// TIA Portal V17 export
// export: Created 2024-08-26T21:07:19.2791777Z, ExportSetting WithDefaults, DisplayName Totally Integrated Automation Portal, DisplayVersion V17 Update 7, DisplayName TIA Portal Openness, DisplayVersion V17 Update 7, DisplayName TIA Portal Version Control Interface, DisplayVersion V17, DisplayName SINAMICS Startdrive Advanced, DisplayVersion V17 SP2, DisplayName SINAMICS Startdrive G110M, G120, G120C, G120D, G120P, G115D, DisplayVersion V17 SP2, DisplayName SINAMICS Startdrive G130, G150, S120, S150, SINAMICS MV, S210, DisplayVersion V17 SP2, DisplayName STEP 7 Professional, DisplayVersion V17 Update 7, DisplayName STEP 7 Safety, DisplayVersion V17 Update 6, DisplayName WinCC Advanced / Unified PC, DisplayVersion V17 Update 7
FUNCTION "DINT TO BOOL" : Void   // FC10, LAD
{ S7_Optimized_Access := 'TRUE' }
VERSION : 0.1
// stored: AutoNumber true, IsIECCheckEnabled false, SetENOAutomatically false, UDAEnableTagReadback false
BEGIN

REGION Network 1: A INPUTS STATUS
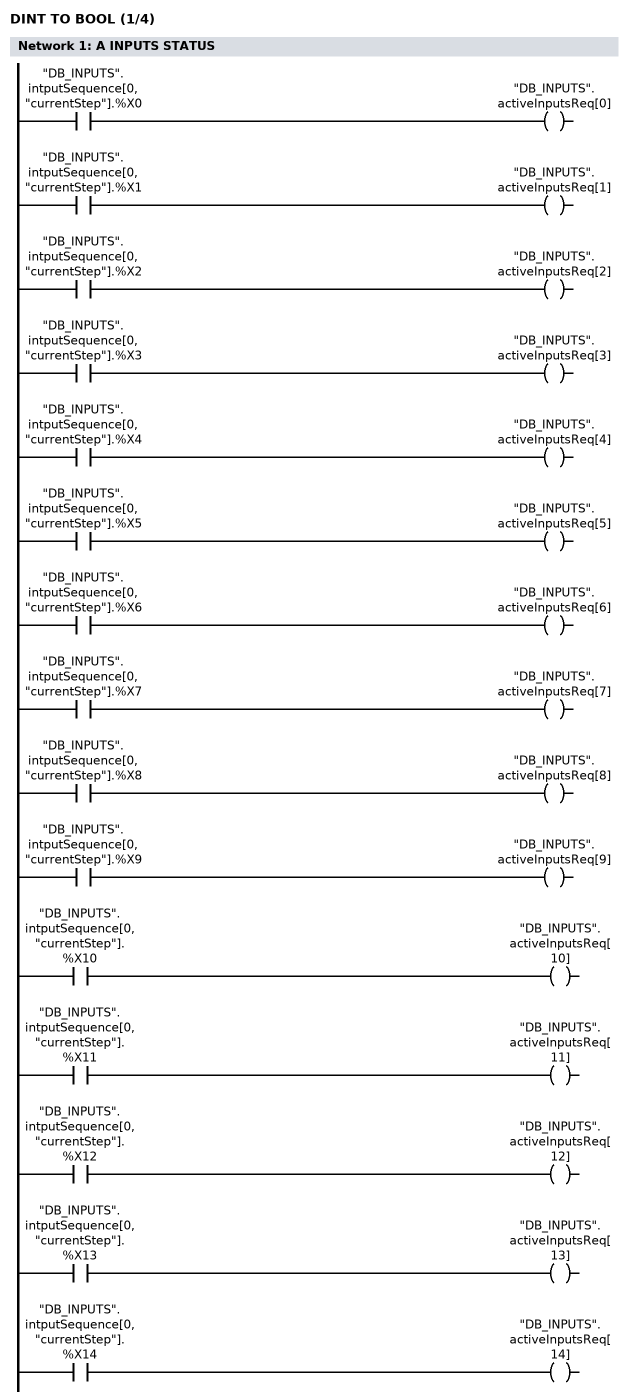
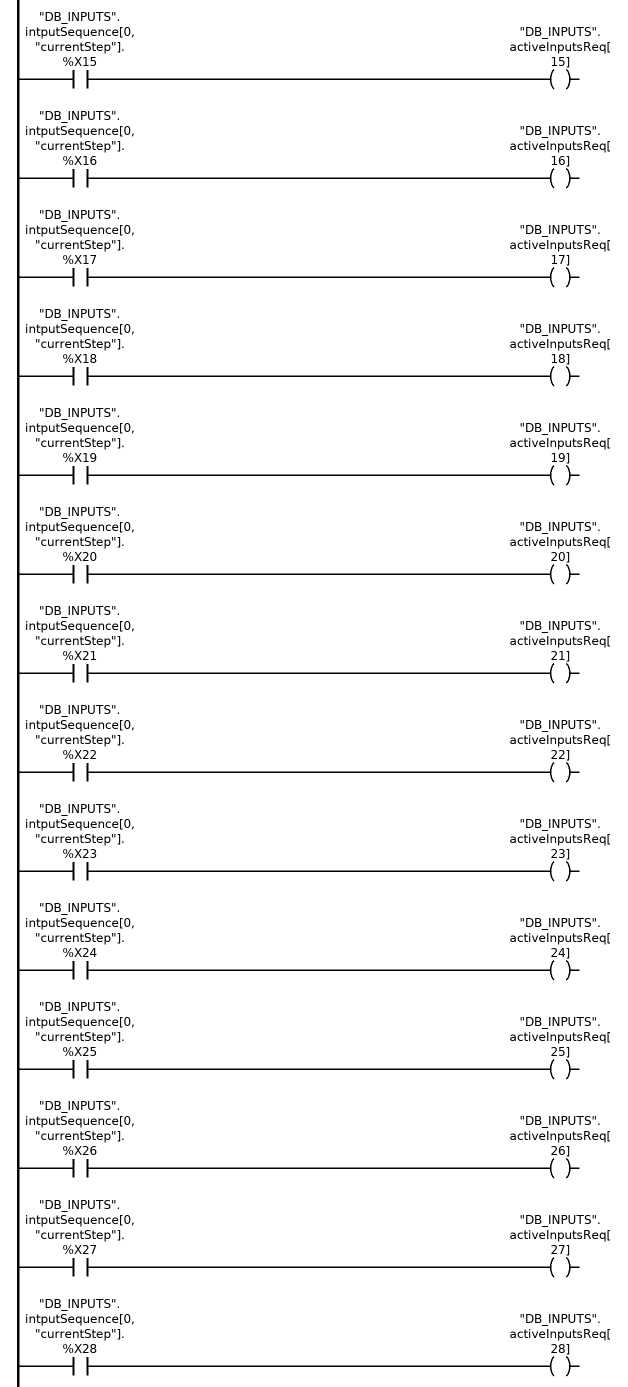
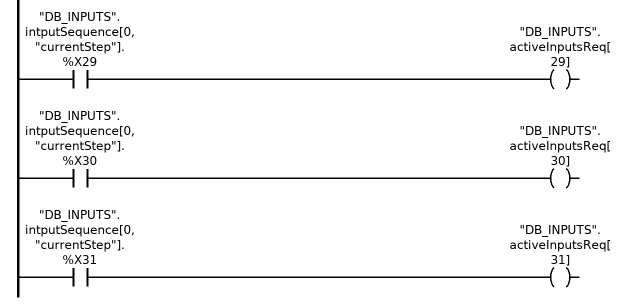
   RUNG wire#powerrail
      Contact( "DB_INPUTS".intputSequence[0, "currentStep"].%X0 )
      Coil( "DB_INPUTS".activeInputsReq[0] )
   END_RUNG
   RUNG wire#powerrail
      Contact( "DB_INPUTS".intputSequence[0, "currentStep"].%X1 )
      Coil( "DB_INPUTS".activeInputsReq[1] )
   END_RUNG
   RUNG wire#powerrail
      Contact( "DB_INPUTS".intputSequence[0, "currentStep"].%X2 )
      Coil( "DB_INPUTS".activeInputsReq[2] )
   END_RUNG
   RUNG wire#powerrail
      Contact( "DB_INPUTS".intputSequence[0, "currentStep"].%X3 )
      Coil( "DB_INPUTS".activeInputsReq[3] )
   END_RUNG
   RUNG wire#powerrail
      Contact( "DB_INPUTS".intputSequence[0, "currentStep"].%X4 )
      Coil( "DB_INPUTS".activeInputsReq[4] )
   END_RUNG
   RUNG wire#powerrail
      Contact( "DB_INPUTS".intputSequence[0, "currentStep"].%X5 )
      Coil( "DB_INPUTS".activeInputsReq[5] )
   END_RUNG
   RUNG wire#powerrail
      Contact( "DB_INPUTS".intputSequence[0, "currentStep"].%X6 )
      Coil( "DB_INPUTS".activeInputsReq[6] )
   END_RUNG
   RUNG wire#powerrail
      Contact( "DB_INPUTS".intputSequence[0, "currentStep"].%X7 )
      Coil( "DB_INPUTS".activeInputsReq[7] )
   END_RUNG
   RUNG wire#powerrail
      Contact( "DB_INPUTS".intputSequence[0, "currentStep"].%X8 )
      Coil( "DB_INPUTS".activeInputsReq[8] )
   END_RUNG
   RUNG wire#powerrail
      Contact( "DB_INPUTS".intputSequence[0, "currentStep"].%X9 )
      Coil( "DB_INPUTS".activeInputsReq[9] )
   END_RUNG
   RUNG wire#powerrail
      Contact( "DB_INPUTS".intputSequence[0, "currentStep"].%X10 )
      Coil( "DB_INPUTS".activeInputsReq[10] )
   END_RUNG
   RUNG wire#powerrail
      Contact( "DB_INPUTS".intputSequence[0, "currentStep"].%X11 )
      Coil( "DB_INPUTS".activeInputsReq[11] )
   END_RUNG
   RUNG wire#powerrail
      Contact( "DB_INPUTS".intputSequence[0, "currentStep"].%X12 )
      Coil( "DB_INPUTS".activeInputsReq[12] )
   END_RUNG
   RUNG wire#powerrail
      Contact( "DB_INPUTS".intputSequence[0, "currentStep"].%X13 )
      Coil( "DB_INPUTS".activeInputsReq[13] )
   END_RUNG
   RUNG wire#powerrail
      Contact( "DB_INPUTS".intputSequence[0, "currentStep"].%X14 )
      Coil( "DB_INPUTS".activeInputsReq[14] )
   END_RUNG
   RUNG wire#powerrail
      Contact( "DB_INPUTS".intputSequence[0, "currentStep"].%X15 )
      Coil( "DB_INPUTS".activeInputsReq[15] )
   END_RUNG
   RUNG wire#powerrail
      Contact( "DB_INPUTS".intputSequence[0, "currentStep"].%X16 )
      Coil( "DB_INPUTS".activeInputsReq[16] )
   END_RUNG
   RUNG wire#powerrail
      Contact( "DB_INPUTS".intputSequence[0, "currentStep"].%X17 )
      Coil( "DB_INPUTS".activeInputsReq[17] )
   END_RUNG
   RUNG wire#powerrail
      Contact( "DB_INPUTS".intputSequence[0, "currentStep"].%X18 )
      Coil( "DB_INPUTS".activeInputsReq[18] )
   END_RUNG
   RUNG wire#powerrail
      Contact( "DB_INPUTS".intputSequence[0, "currentStep"].%X19 )
      Coil( "DB_INPUTS".activeInputsReq[19] )
   END_RUNG
   RUNG wire#powerrail
      Contact( "DB_INPUTS".intputSequence[0, "currentStep"].%X20 )
      Coil( "DB_INPUTS".activeInputsReq[20] )
   END_RUNG
   RUNG wire#powerrail
      Contact( "DB_INPUTS".intputSequence[0, "currentStep"].%X21 )
      Coil( "DB_INPUTS".activeInputsReq[21] )
   END_RUNG
   RUNG wire#powerrail
      Contact( "DB_INPUTS".intputSequence[0, "currentStep"].%X22 )
      Coil( "DB_INPUTS".activeInputsReq[22] )
   END_RUNG
   RUNG wire#powerrail
      Contact( "DB_INPUTS".intputSequence[0, "currentStep"].%X23 )
      Coil( "DB_INPUTS".activeInputsReq[23] )
   END_RUNG
   RUNG wire#powerrail
      Contact( "DB_INPUTS".intputSequence[0, "currentStep"].%X24 )
      Coil( "DB_INPUTS".activeInputsReq[24] )
   END_RUNG
   RUNG wire#powerrail
      Contact( "DB_INPUTS".intputSequence[0, "currentStep"].%X25 )
      Coil( "DB_INPUTS".activeInputsReq[25] )
   END_RUNG
   RUNG wire#powerrail
      Contact( "DB_INPUTS".intputSequence[0, "currentStep"].%X26 )
      Coil( "DB_INPUTS".activeInputsReq[26] )
   END_RUNG
   RUNG wire#powerrail
      Contact( "DB_INPUTS".intputSequence[0, "currentStep"].%X27 )
      Coil( "DB_INPUTS".activeInputsReq[27] )
   END_RUNG
   RUNG wire#powerrail
      Contact( "DB_INPUTS".intputSequence[0, "currentStep"].%X28 )
      Coil( "DB_INPUTS".activeInputsReq[28] )
   END_RUNG
   RUNG wire#powerrail
      Contact( "DB_INPUTS".intputSequence[0, "currentStep"].%X29 )
      Coil( "DB_INPUTS".activeInputsReq[29] )
   END_RUNG
   RUNG wire#powerrail
      Contact( "DB_INPUTS".intputSequence[0, "currentStep"].%X30 )
      Coil( "DB_INPUTS".activeInputsReq[30] )
   END_RUNG
   RUNG wire#powerrail
      Contact( "DB_INPUTS".intputSequence[0, "currentStep"].%X31 )
      Coil( "DB_INPUTS".activeInputsReq[31] )
   END_RUNG
   // the same network as SCL:
   "DB_INPUTS".activeInputsReq[0] := "DB_INPUTS".intputSequence[0, "currentStep"].%X0;
   "DB_INPUTS".activeInputsReq[1] := "DB_INPUTS".intputSequence[0, "currentStep"].%X1;
   "DB_INPUTS".activeInputsReq[2] := "DB_INPUTS".intputSequence[0, "currentStep"].%X2;
   "DB_INPUTS".activeInputsReq[3] := "DB_INPUTS".intputSequence[0, "currentStep"].%X3;
   "DB_INPUTS".activeInputsReq[4] := "DB_INPUTS".intputSequence[0, "currentStep"].%X4;
   "DB_INPUTS".activeInputsReq[5] := "DB_INPUTS".intputSequence[0, "currentStep"].%X5;
   "DB_INPUTS".activeInputsReq[6] := "DB_INPUTS".intputSequence[0, "currentStep"].%X6;
   "DB_INPUTS".activeInputsReq[7] := "DB_INPUTS".intputSequence[0, "currentStep"].%X7;
   "DB_INPUTS".activeInputsReq[8] := "DB_INPUTS".intputSequence[0, "currentStep"].%X8;
   "DB_INPUTS".activeInputsReq[9] := "DB_INPUTS".intputSequence[0, "currentStep"].%X9;
   "DB_INPUTS".activeInputsReq[10] := "DB_INPUTS".intputSequence[0, "currentStep"].%X10;
   "DB_INPUTS".activeInputsReq[11] := "DB_INPUTS".intputSequence[0, "currentStep"].%X11;
   "DB_INPUTS".activeInputsReq[12] := "DB_INPUTS".intputSequence[0, "currentStep"].%X12;
   "DB_INPUTS".activeInputsReq[13] := "DB_INPUTS".intputSequence[0, "currentStep"].%X13;
   "DB_INPUTS".activeInputsReq[14] := "DB_INPUTS".intputSequence[0, "currentStep"].%X14;
   "DB_INPUTS".activeInputsReq[15] := "DB_INPUTS".intputSequence[0, "currentStep"].%X15;
   "DB_INPUTS".activeInputsReq[16] := "DB_INPUTS".intputSequence[0, "currentStep"].%X16;
   "DB_INPUTS".activeInputsReq[17] := "DB_INPUTS".intputSequence[0, "currentStep"].%X17;
   "DB_INPUTS".activeInputsReq[18] := "DB_INPUTS".intputSequence[0, "currentStep"].%X18;
   "DB_INPUTS".activeInputsReq[19] := "DB_INPUTS".intputSequence[0, "currentStep"].%X19;
   "DB_INPUTS".activeInputsReq[20] := "DB_INPUTS".intputSequence[0, "currentStep"].%X20;
   "DB_INPUTS".activeInputsReq[21] := "DB_INPUTS".intputSequence[0, "currentStep"].%X21;
   "DB_INPUTS".activeInputsReq[22] := "DB_INPUTS".intputSequence[0, "currentStep"].%X22;
   "DB_INPUTS".activeInputsReq[23] := "DB_INPUTS".intputSequence[0, "currentStep"].%X23;
   "DB_INPUTS".activeInputsReq[24] := "DB_INPUTS".intputSequence[0, "currentStep"].%X24;
   "DB_INPUTS".activeInputsReq[25] := "DB_INPUTS".intputSequence[0, "currentStep"].%X25;
   "DB_INPUTS".activeInputsReq[26] := "DB_INPUTS".intputSequence[0, "currentStep"].%X26;
   "DB_INPUTS".activeInputsReq[27] := "DB_INPUTS".intputSequence[0, "currentStep"].%X27;
   "DB_INPUTS".activeInputsReq[28] := "DB_INPUTS".intputSequence[0, "currentStep"].%X28;
   "DB_INPUTS".activeInputsReq[29] := "DB_INPUTS".intputSequence[0, "currentStep"].%X29;
   "DB_INPUTS".activeInputsReq[30] := "DB_INPUTS".intputSequence[0, "currentStep"].%X30;
   "DB_INPUTS".activeInputsReq[31] := "DB_INPUTS".intputSequence[0, "currentStep"].%X31;
END_REGION

REGION Network 2: MASK INPUTS STATUS
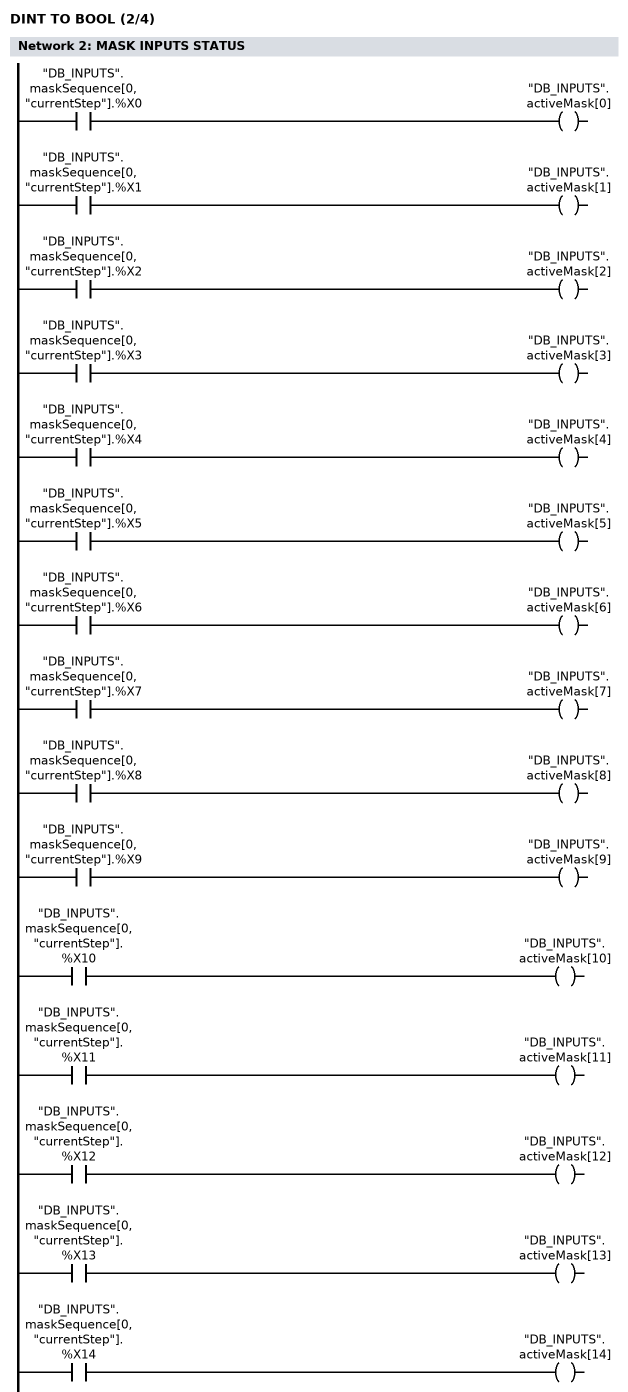
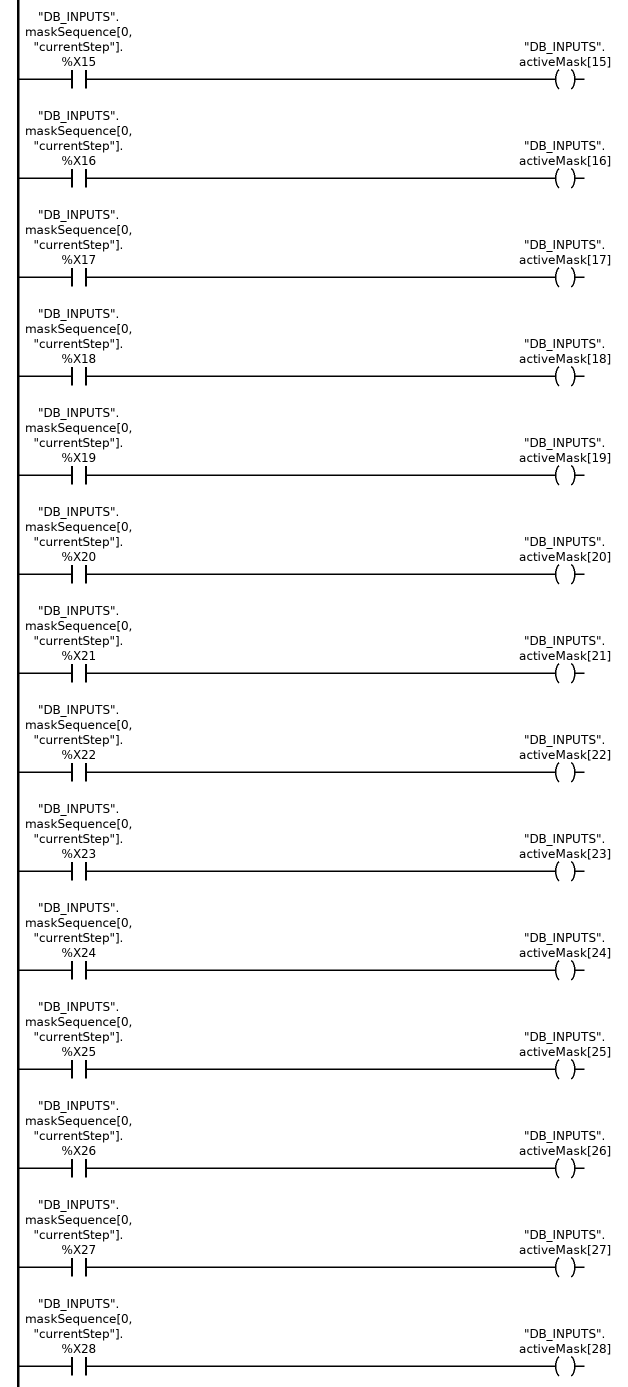
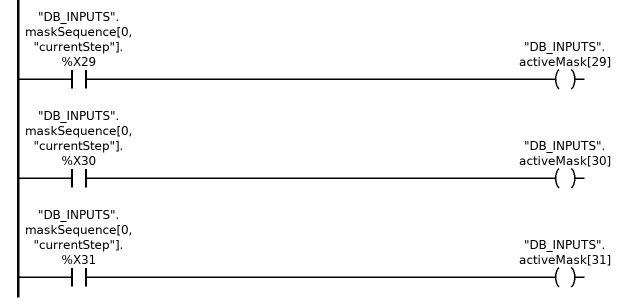
   RUNG wire#powerrail
      Contact( "DB_INPUTS".maskSequence[0, "currentStep"].%X0 )
      Coil( "DB_INPUTS".activeMask[0] )
   END_RUNG
   RUNG wire#powerrail
      Contact( "DB_INPUTS".maskSequence[0, "currentStep"].%X1 )
      Coil( "DB_INPUTS".activeMask[1] )
   END_RUNG
   RUNG wire#powerrail
      Contact( "DB_INPUTS".maskSequence[0, "currentStep"].%X2 )
      Coil( "DB_INPUTS".activeMask[2] )
   END_RUNG
   RUNG wire#powerrail
      Contact( "DB_INPUTS".maskSequence[0, "currentStep"].%X3 )
      Coil( "DB_INPUTS".activeMask[3] )
   END_RUNG
   RUNG wire#powerrail
      Contact( "DB_INPUTS".maskSequence[0, "currentStep"].%X4 )
      Coil( "DB_INPUTS".activeMask[4] )
   END_RUNG
   RUNG wire#powerrail
      Contact( "DB_INPUTS".maskSequence[0, "currentStep"].%X5 )
      Coil( "DB_INPUTS".activeMask[5] )
   END_RUNG
   RUNG wire#powerrail
      Contact( "DB_INPUTS".maskSequence[0, "currentStep"].%X6 )
      Coil( "DB_INPUTS".activeMask[6] )
   END_RUNG
   RUNG wire#powerrail
      Contact( "DB_INPUTS".maskSequence[0, "currentStep"].%X7 )
      Coil( "DB_INPUTS".activeMask[7] )
   END_RUNG
   RUNG wire#powerrail
      Contact( "DB_INPUTS".maskSequence[0, "currentStep"].%X8 )
      Coil( "DB_INPUTS".activeMask[8] )
   END_RUNG
   RUNG wire#powerrail
      Contact( "DB_INPUTS".maskSequence[0, "currentStep"].%X9 )
      Coil( "DB_INPUTS".activeMask[9] )
   END_RUNG
   RUNG wire#powerrail
      Contact( "DB_INPUTS".maskSequence[0, "currentStep"].%X10 )
      Coil( "DB_INPUTS".activeMask[10] )
   END_RUNG
   RUNG wire#powerrail
      Contact( "DB_INPUTS".maskSequence[0, "currentStep"].%X11 )
      Coil( "DB_INPUTS".activeMask[11] )
   END_RUNG
   RUNG wire#powerrail
      Contact( "DB_INPUTS".maskSequence[0, "currentStep"].%X12 )
      Coil( "DB_INPUTS".activeMask[12] )
   END_RUNG
   RUNG wire#powerrail
      Contact( "DB_INPUTS".maskSequence[0, "currentStep"].%X13 )
      Coil( "DB_INPUTS".activeMask[13] )
   END_RUNG
   RUNG wire#powerrail
      Contact( "DB_INPUTS".maskSequence[0, "currentStep"].%X14 )
      Coil( "DB_INPUTS".activeMask[14] )
   END_RUNG
   RUNG wire#powerrail
      Contact( "DB_INPUTS".maskSequence[0, "currentStep"].%X15 )
      Coil( "DB_INPUTS".activeMask[15] )
   END_RUNG
   RUNG wire#powerrail
      Contact( "DB_INPUTS".maskSequence[0, "currentStep"].%X16 )
      Coil( "DB_INPUTS".activeMask[16] )
   END_RUNG
   RUNG wire#powerrail
      Contact( "DB_INPUTS".maskSequence[0, "currentStep"].%X17 )
      Coil( "DB_INPUTS".activeMask[17] )
   END_RUNG
   RUNG wire#powerrail
      Contact( "DB_INPUTS".maskSequence[0, "currentStep"].%X18 )
      Coil( "DB_INPUTS".activeMask[18] )
   END_RUNG
   RUNG wire#powerrail
      Contact( "DB_INPUTS".maskSequence[0, "currentStep"].%X19 )
      Coil( "DB_INPUTS".activeMask[19] )
   END_RUNG
   RUNG wire#powerrail
      Contact( "DB_INPUTS".maskSequence[0, "currentStep"].%X20 )
      Coil( "DB_INPUTS".activeMask[20] )
   END_RUNG
   RUNG wire#powerrail
      Contact( "DB_INPUTS".maskSequence[0, "currentStep"].%X21 )
      Coil( "DB_INPUTS".activeMask[21] )
   END_RUNG
   RUNG wire#powerrail
      Contact( "DB_INPUTS".maskSequence[0, "currentStep"].%X22 )
      Coil( "DB_INPUTS".activeMask[22] )
   END_RUNG
   RUNG wire#powerrail
      Contact( "DB_INPUTS".maskSequence[0, "currentStep"].%X23 )
      Coil( "DB_INPUTS".activeMask[23] )
   END_RUNG
   RUNG wire#powerrail
      Contact( "DB_INPUTS".maskSequence[0, "currentStep"].%X24 )
      Coil( "DB_INPUTS".activeMask[24] )
   END_RUNG
   RUNG wire#powerrail
      Contact( "DB_INPUTS".maskSequence[0, "currentStep"].%X25 )
      Coil( "DB_INPUTS".activeMask[25] )
   END_RUNG
   RUNG wire#powerrail
      Contact( "DB_INPUTS".maskSequence[0, "currentStep"].%X26 )
      Coil( "DB_INPUTS".activeMask[26] )
   END_RUNG
   RUNG wire#powerrail
      Contact( "DB_INPUTS".maskSequence[0, "currentStep"].%X27 )
      Coil( "DB_INPUTS".activeMask[27] )
   END_RUNG
   RUNG wire#powerrail
      Contact( "DB_INPUTS".maskSequence[0, "currentStep"].%X28 )
      Coil( "DB_INPUTS".activeMask[28] )
   END_RUNG
   RUNG wire#powerrail
      Contact( "DB_INPUTS".maskSequence[0, "currentStep"].%X29 )
      Coil( "DB_INPUTS".activeMask[29] )
   END_RUNG
   RUNG wire#powerrail
      Contact( "DB_INPUTS".maskSequence[0, "currentStep"].%X30 )
      Coil( "DB_INPUTS".activeMask[30] )
   END_RUNG
   RUNG wire#powerrail
      Contact( "DB_INPUTS".maskSequence[0, "currentStep"].%X31 )
      Coil( "DB_INPUTS".activeMask[31] )
   END_RUNG
   // the same network as SCL:
   "DB_INPUTS".activeMask[0] := "DB_INPUTS".maskSequence[0, "currentStep"].%X0;
   "DB_INPUTS".activeMask[1] := "DB_INPUTS".maskSequence[0, "currentStep"].%X1;
   "DB_INPUTS".activeMask[2] := "DB_INPUTS".maskSequence[0, "currentStep"].%X2;
   "DB_INPUTS".activeMask[3] := "DB_INPUTS".maskSequence[0, "currentStep"].%X3;
   "DB_INPUTS".activeMask[4] := "DB_INPUTS".maskSequence[0, "currentStep"].%X4;
   "DB_INPUTS".activeMask[5] := "DB_INPUTS".maskSequence[0, "currentStep"].%X5;
   "DB_INPUTS".activeMask[6] := "DB_INPUTS".maskSequence[0, "currentStep"].%X6;
   "DB_INPUTS".activeMask[7] := "DB_INPUTS".maskSequence[0, "currentStep"].%X7;
   "DB_INPUTS".activeMask[8] := "DB_INPUTS".maskSequence[0, "currentStep"].%X8;
   "DB_INPUTS".activeMask[9] := "DB_INPUTS".maskSequence[0, "currentStep"].%X9;
   "DB_INPUTS".activeMask[10] := "DB_INPUTS".maskSequence[0, "currentStep"].%X10;
   "DB_INPUTS".activeMask[11] := "DB_INPUTS".maskSequence[0, "currentStep"].%X11;
   "DB_INPUTS".activeMask[12] := "DB_INPUTS".maskSequence[0, "currentStep"].%X12;
   "DB_INPUTS".activeMask[13] := "DB_INPUTS".maskSequence[0, "currentStep"].%X13;
   "DB_INPUTS".activeMask[14] := "DB_INPUTS".maskSequence[0, "currentStep"].%X14;
   "DB_INPUTS".activeMask[15] := "DB_INPUTS".maskSequence[0, "currentStep"].%X15;
   "DB_INPUTS".activeMask[16] := "DB_INPUTS".maskSequence[0, "currentStep"].%X16;
   "DB_INPUTS".activeMask[17] := "DB_INPUTS".maskSequence[0, "currentStep"].%X17;
   "DB_INPUTS".activeMask[18] := "DB_INPUTS".maskSequence[0, "currentStep"].%X18;
   "DB_INPUTS".activeMask[19] := "DB_INPUTS".maskSequence[0, "currentStep"].%X19;
   "DB_INPUTS".activeMask[20] := "DB_INPUTS".maskSequence[0, "currentStep"].%X20;
   "DB_INPUTS".activeMask[21] := "DB_INPUTS".maskSequence[0, "currentStep"].%X21;
   "DB_INPUTS".activeMask[22] := "DB_INPUTS".maskSequence[0, "currentStep"].%X22;
   "DB_INPUTS".activeMask[23] := "DB_INPUTS".maskSequence[0, "currentStep"].%X23;
   "DB_INPUTS".activeMask[24] := "DB_INPUTS".maskSequence[0, "currentStep"].%X24;
   "DB_INPUTS".activeMask[25] := "DB_INPUTS".maskSequence[0, "currentStep"].%X25;
   "DB_INPUTS".activeMask[26] := "DB_INPUTS".maskSequence[0, "currentStep"].%X26;
   "DB_INPUTS".activeMask[27] := "DB_INPUTS".maskSequence[0, "currentStep"].%X27;
   "DB_INPUTS".activeMask[28] := "DB_INPUTS".maskSequence[0, "currentStep"].%X28;
   "DB_INPUTS".activeMask[29] := "DB_INPUTS".maskSequence[0, "currentStep"].%X29;
   "DB_INPUTS".activeMask[30] := "DB_INPUTS".maskSequence[0, "currentStep"].%X30;
   "DB_INPUTS".activeMask[31] := "DB_INPUTS".maskSequence[0, "currentStep"].%X31;
END_REGION

REGION Network 3: B OUTPUTS STATUS
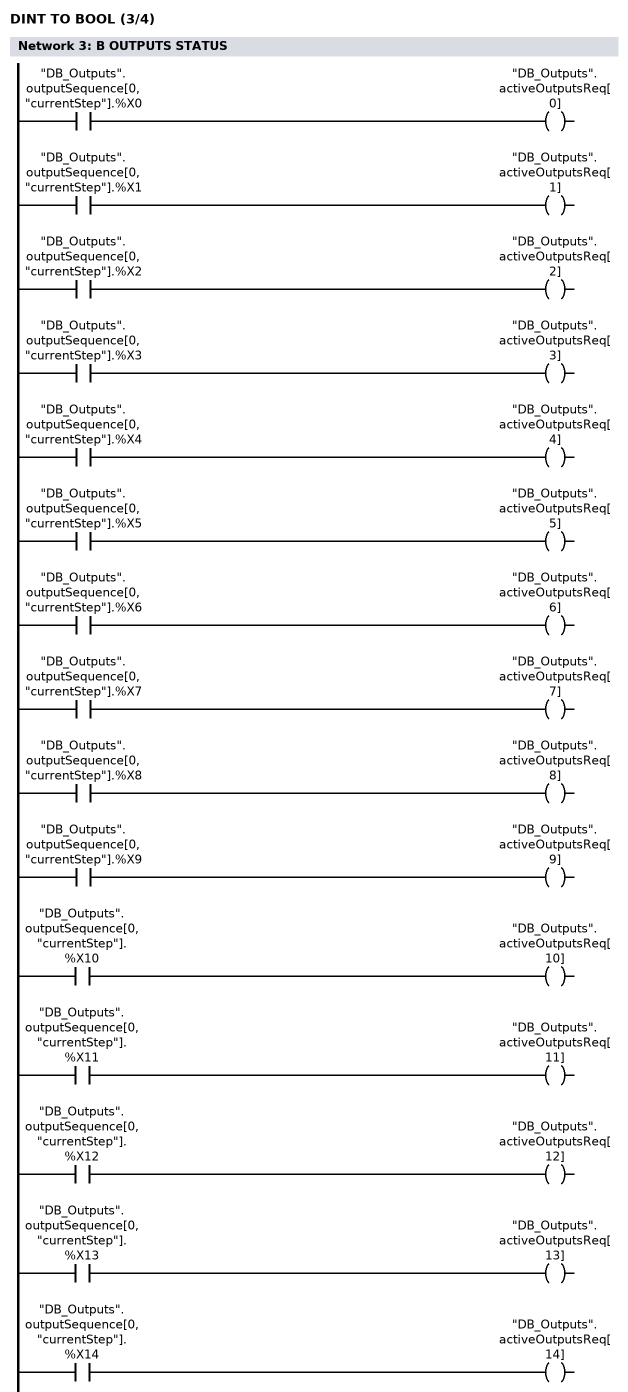
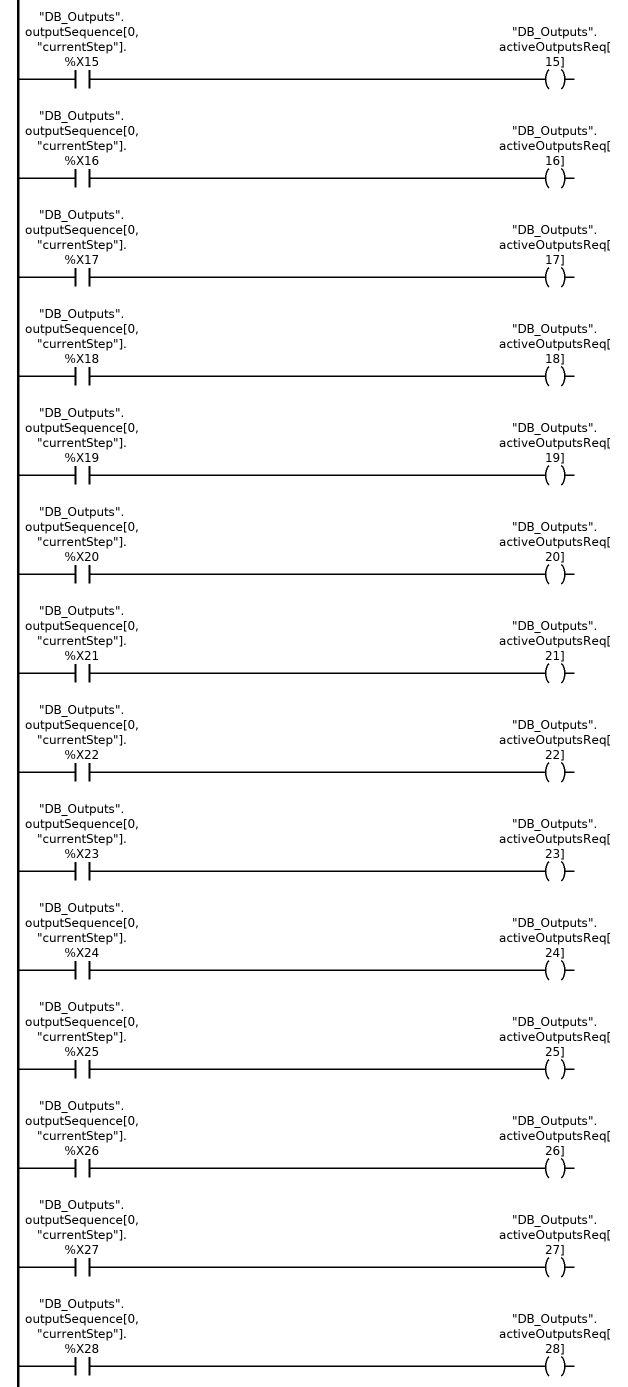
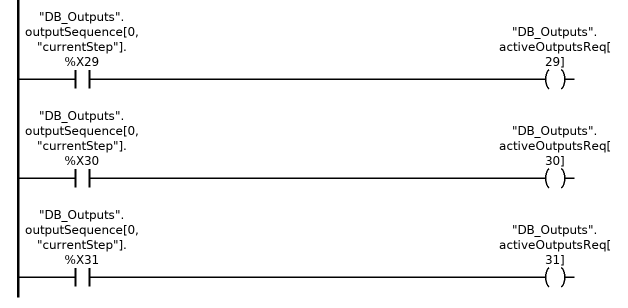
   RUNG wire#powerrail
      Contact( "DB_Outputs".outputSequence[0, "currentStep"].%X0 )
      Coil( "DB_Outputs".activeOutputsReq[0] )
   END_RUNG
   RUNG wire#powerrail
      Contact( "DB_Outputs".outputSequence[0, "currentStep"].%X1 )
      Coil( "DB_Outputs".activeOutputsReq[1] )
   END_RUNG
   RUNG wire#powerrail
      Contact( "DB_Outputs".outputSequence[0, "currentStep"].%X2 )
      Coil( "DB_Outputs".activeOutputsReq[2] )
   END_RUNG
   RUNG wire#powerrail
      Contact( "DB_Outputs".outputSequence[0, "currentStep"].%X3 )
      Coil( "DB_Outputs".activeOutputsReq[3] )
   END_RUNG
   RUNG wire#powerrail
      Contact( "DB_Outputs".outputSequence[0, "currentStep"].%X4 )
      Coil( "DB_Outputs".activeOutputsReq[4] )
   END_RUNG
   RUNG wire#powerrail
      Contact( "DB_Outputs".outputSequence[0, "currentStep"].%X5 )
      Coil( "DB_Outputs".activeOutputsReq[5] )
   END_RUNG
   RUNG wire#powerrail
      Contact( "DB_Outputs".outputSequence[0, "currentStep"].%X6 )
      Coil( "DB_Outputs".activeOutputsReq[6] )
   END_RUNG
   RUNG wire#powerrail
      Contact( "DB_Outputs".outputSequence[0, "currentStep"].%X7 )
      Coil( "DB_Outputs".activeOutputsReq[7] )
   END_RUNG
   RUNG wire#powerrail
      Contact( "DB_Outputs".outputSequence[0, "currentStep"].%X8 )
      Coil( "DB_Outputs".activeOutputsReq[8] )
   END_RUNG
   RUNG wire#powerrail
      Contact( "DB_Outputs".outputSequence[0, "currentStep"].%X9 )
      Coil( "DB_Outputs".activeOutputsReq[9] )
   END_RUNG
   RUNG wire#powerrail
      Contact( "DB_Outputs".outputSequence[0, "currentStep"].%X10 )
      Coil( "DB_Outputs".activeOutputsReq[10] )
   END_RUNG
   RUNG wire#powerrail
      Contact( "DB_Outputs".outputSequence[0, "currentStep"].%X11 )
      Coil( "DB_Outputs".activeOutputsReq[11] )
   END_RUNG
   RUNG wire#powerrail
      Contact( "DB_Outputs".outputSequence[0, "currentStep"].%X12 )
      Coil( "DB_Outputs".activeOutputsReq[12] )
   END_RUNG
   RUNG wire#powerrail
      Contact( "DB_Outputs".outputSequence[0, "currentStep"].%X13 )
      Coil( "DB_Outputs".activeOutputsReq[13] )
   END_RUNG
   RUNG wire#powerrail
      Contact( "DB_Outputs".outputSequence[0, "currentStep"].%X14 )
      Coil( "DB_Outputs".activeOutputsReq[14] )
   END_RUNG
   RUNG wire#powerrail
      Contact( "DB_Outputs".outputSequence[0, "currentStep"].%X15 )
      Coil( "DB_Outputs".activeOutputsReq[15] )
   END_RUNG
   RUNG wire#powerrail
      Contact( "DB_Outputs".outputSequence[0, "currentStep"].%X16 )
      Coil( "DB_Outputs".activeOutputsReq[16] )
   END_RUNG
   RUNG wire#powerrail
      Contact( "DB_Outputs".outputSequence[0, "currentStep"].%X17 )
      Coil( "DB_Outputs".activeOutputsReq[17] )
   END_RUNG
   RUNG wire#powerrail
      Contact( "DB_Outputs".outputSequence[0, "currentStep"].%X18 )
      Coil( "DB_Outputs".activeOutputsReq[18] )
   END_RUNG
   RUNG wire#powerrail
      Contact( "DB_Outputs".outputSequence[0, "currentStep"].%X19 )
      Coil( "DB_Outputs".activeOutputsReq[19] )
   END_RUNG
   RUNG wire#powerrail
      Contact( "DB_Outputs".outputSequence[0, "currentStep"].%X20 )
      Coil( "DB_Outputs".activeOutputsReq[20] )
   END_RUNG
   RUNG wire#powerrail
      Contact( "DB_Outputs".outputSequence[0, "currentStep"].%X21 )
      Coil( "DB_Outputs".activeOutputsReq[21] )
   END_RUNG
   RUNG wire#powerrail
      Contact( "DB_Outputs".outputSequence[0, "currentStep"].%X22 )
      Coil( "DB_Outputs".activeOutputsReq[22] )
   END_RUNG
   RUNG wire#powerrail
      Contact( "DB_Outputs".outputSequence[0, "currentStep"].%X23 )
      Coil( "DB_Outputs".activeOutputsReq[23] )
   END_RUNG
   RUNG wire#powerrail
      Contact( "DB_Outputs".outputSequence[0, "currentStep"].%X24 )
      Coil( "DB_Outputs".activeOutputsReq[24] )
   END_RUNG
   RUNG wire#powerrail
      Contact( "DB_Outputs".outputSequence[0, "currentStep"].%X25 )
      Coil( "DB_Outputs".activeOutputsReq[25] )
   END_RUNG
   RUNG wire#powerrail
      Contact( "DB_Outputs".outputSequence[0, "currentStep"].%X26 )
      Coil( "DB_Outputs".activeOutputsReq[26] )
   END_RUNG
   RUNG wire#powerrail
      Contact( "DB_Outputs".outputSequence[0, "currentStep"].%X27 )
      Coil( "DB_Outputs".activeOutputsReq[27] )
   END_RUNG
   RUNG wire#powerrail
      Contact( "DB_Outputs".outputSequence[0, "currentStep"].%X28 )
      Coil( "DB_Outputs".activeOutputsReq[28] )
   END_RUNG
   RUNG wire#powerrail
      Contact( "DB_Outputs".outputSequence[0, "currentStep"].%X29 )
      Coil( "DB_Outputs".activeOutputsReq[29] )
   END_RUNG
   RUNG wire#powerrail
      Contact( "DB_Outputs".outputSequence[0, "currentStep"].%X30 )
      Coil( "DB_Outputs".activeOutputsReq[30] )
   END_RUNG
   RUNG wire#powerrail
      Contact( "DB_Outputs".outputSequence[0, "currentStep"].%X31 )
      Coil( "DB_Outputs".activeOutputsReq[31] )
   END_RUNG
   // the same network as SCL:
   "DB_Outputs".activeOutputsReq[0] := "DB_Outputs".outputSequence[0, "currentStep"].%X0;
   "DB_Outputs".activeOutputsReq[1] := "DB_Outputs".outputSequence[0, "currentStep"].%X1;
   "DB_Outputs".activeOutputsReq[2] := "DB_Outputs".outputSequence[0, "currentStep"].%X2;
   "DB_Outputs".activeOutputsReq[3] := "DB_Outputs".outputSequence[0, "currentStep"].%X3;
   "DB_Outputs".activeOutputsReq[4] := "DB_Outputs".outputSequence[0, "currentStep"].%X4;
   "DB_Outputs".activeOutputsReq[5] := "DB_Outputs".outputSequence[0, "currentStep"].%X5;
   "DB_Outputs".activeOutputsReq[6] := "DB_Outputs".outputSequence[0, "currentStep"].%X6;
   "DB_Outputs".activeOutputsReq[7] := "DB_Outputs".outputSequence[0, "currentStep"].%X7;
   "DB_Outputs".activeOutputsReq[8] := "DB_Outputs".outputSequence[0, "currentStep"].%X8;
   "DB_Outputs".activeOutputsReq[9] := "DB_Outputs".outputSequence[0, "currentStep"].%X9;
   "DB_Outputs".activeOutputsReq[10] := "DB_Outputs".outputSequence[0, "currentStep"].%X10;
   "DB_Outputs".activeOutputsReq[11] := "DB_Outputs".outputSequence[0, "currentStep"].%X11;
   "DB_Outputs".activeOutputsReq[12] := "DB_Outputs".outputSequence[0, "currentStep"].%X12;
   "DB_Outputs".activeOutputsReq[13] := "DB_Outputs".outputSequence[0, "currentStep"].%X13;
   "DB_Outputs".activeOutputsReq[14] := "DB_Outputs".outputSequence[0, "currentStep"].%X14;
   "DB_Outputs".activeOutputsReq[15] := "DB_Outputs".outputSequence[0, "currentStep"].%X15;
   "DB_Outputs".activeOutputsReq[16] := "DB_Outputs".outputSequence[0, "currentStep"].%X16;
   "DB_Outputs".activeOutputsReq[17] := "DB_Outputs".outputSequence[0, "currentStep"].%X17;
   "DB_Outputs".activeOutputsReq[18] := "DB_Outputs".outputSequence[0, "currentStep"].%X18;
   "DB_Outputs".activeOutputsReq[19] := "DB_Outputs".outputSequence[0, "currentStep"].%X19;
   "DB_Outputs".activeOutputsReq[20] := "DB_Outputs".outputSequence[0, "currentStep"].%X20;
   "DB_Outputs".activeOutputsReq[21] := "DB_Outputs".outputSequence[0, "currentStep"].%X21;
   "DB_Outputs".activeOutputsReq[22] := "DB_Outputs".outputSequence[0, "currentStep"].%X22;
   "DB_Outputs".activeOutputsReq[23] := "DB_Outputs".outputSequence[0, "currentStep"].%X23;
   "DB_Outputs".activeOutputsReq[24] := "DB_Outputs".outputSequence[0, "currentStep"].%X24;
   "DB_Outputs".activeOutputsReq[25] := "DB_Outputs".outputSequence[0, "currentStep"].%X25;
   "DB_Outputs".activeOutputsReq[26] := "DB_Outputs".outputSequence[0, "currentStep"].%X26;
   "DB_Outputs".activeOutputsReq[27] := "DB_Outputs".outputSequence[0, "currentStep"].%X27;
   "DB_Outputs".activeOutputsReq[28] := "DB_Outputs".outputSequence[0, "currentStep"].%X28;
   "DB_Outputs".activeOutputsReq[29] := "DB_Outputs".outputSequence[0, "currentStep"].%X29;
   "DB_Outputs".activeOutputsReq[30] := "DB_Outputs".outputSequence[0, "currentStep"].%X30;
   "DB_Outputs".activeOutputsReq[31] := "DB_Outputs".outputSequence[0, "currentStep"].%X31;
END_REGION

REGION Network 4: MASK OUTPUTS STATUS
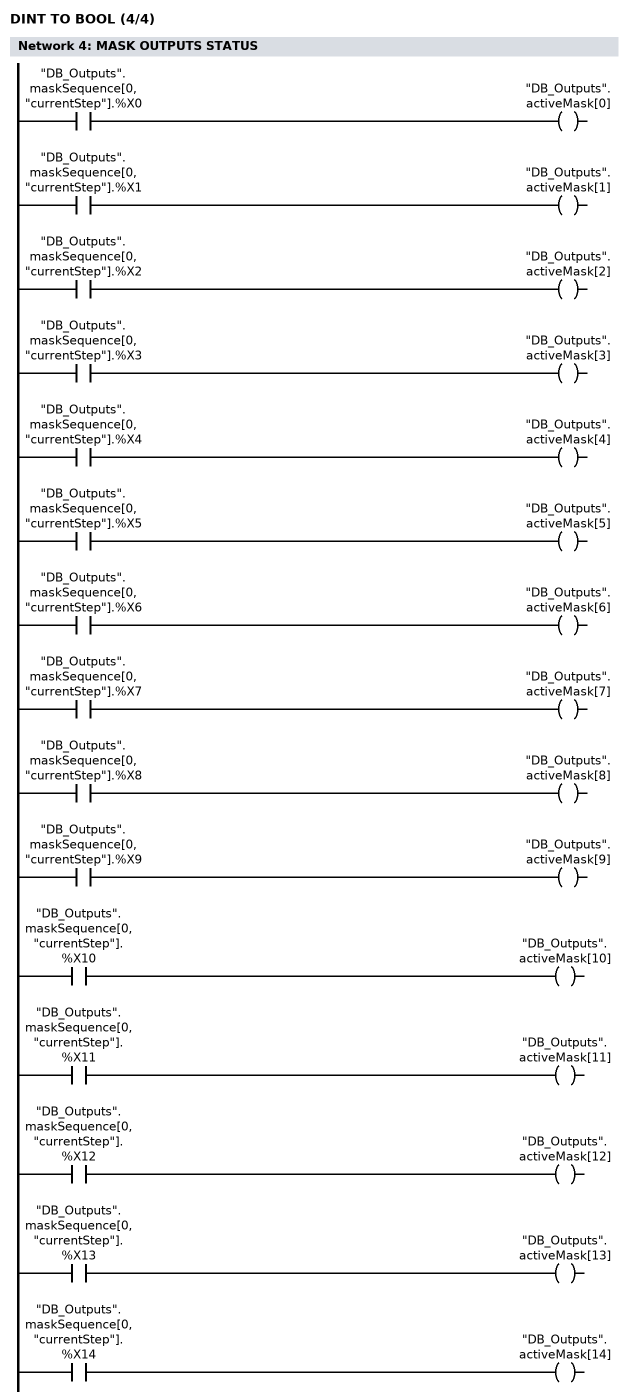
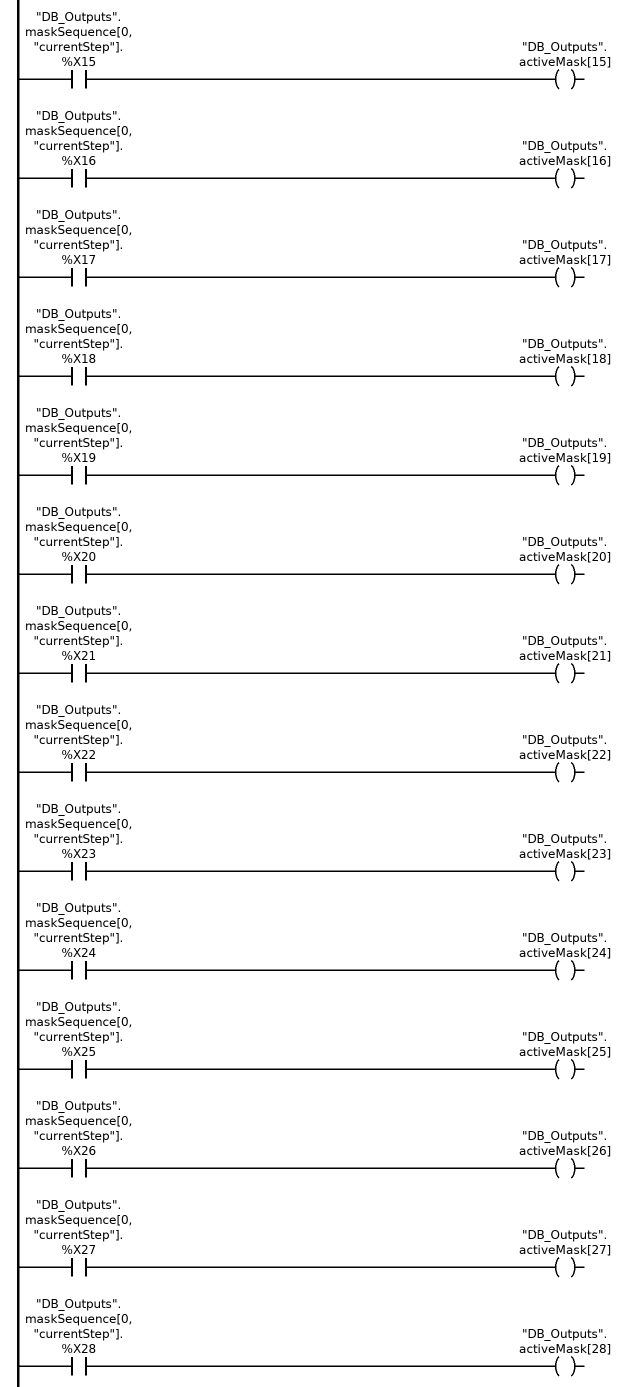
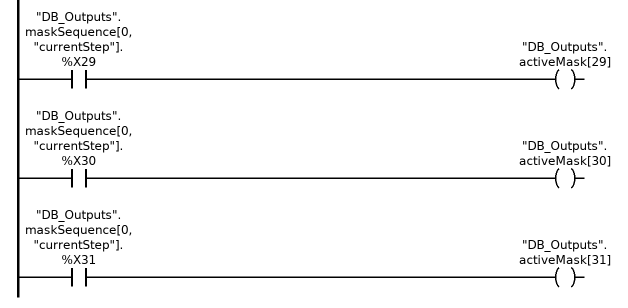
   RUNG wire#powerrail
      Contact( "DB_Outputs".maskSequence[0, "currentStep"].%X0 )
      Coil( "DB_Outputs".activeMask[0] )
   END_RUNG
   RUNG wire#powerrail
      Contact( "DB_Outputs".maskSequence[0, "currentStep"].%X1 )
      Coil( "DB_Outputs".activeMask[1] )
   END_RUNG
   RUNG wire#powerrail
      Contact( "DB_Outputs".maskSequence[0, "currentStep"].%X2 )
      Coil( "DB_Outputs".activeMask[2] )
   END_RUNG
   RUNG wire#powerrail
      Contact( "DB_Outputs".maskSequence[0, "currentStep"].%X3 )
      Coil( "DB_Outputs".activeMask[3] )
   END_RUNG
   RUNG wire#powerrail
      Contact( "DB_Outputs".maskSequence[0, "currentStep"].%X4 )
      Coil( "DB_Outputs".activeMask[4] )
   END_RUNG
   RUNG wire#powerrail
      Contact( "DB_Outputs".maskSequence[0, "currentStep"].%X5 )
      Coil( "DB_Outputs".activeMask[5] )
   END_RUNG
   RUNG wire#powerrail
      Contact( "DB_Outputs".maskSequence[0, "currentStep"].%X6 )
      Coil( "DB_Outputs".activeMask[6] )
   END_RUNG
   RUNG wire#powerrail
      Contact( "DB_Outputs".maskSequence[0, "currentStep"].%X7 )
      Coil( "DB_Outputs".activeMask[7] )
   END_RUNG
   RUNG wire#powerrail
      Contact( "DB_Outputs".maskSequence[0, "currentStep"].%X8 )
      Coil( "DB_Outputs".activeMask[8] )
   END_RUNG
   RUNG wire#powerrail
      Contact( "DB_Outputs".maskSequence[0, "currentStep"].%X9 )
      Coil( "DB_Outputs".activeMask[9] )
   END_RUNG
   RUNG wire#powerrail
      Contact( "DB_Outputs".maskSequence[0, "currentStep"].%X10 )
      Coil( "DB_Outputs".activeMask[10] )
   END_RUNG
   RUNG wire#powerrail
      Contact( "DB_Outputs".maskSequence[0, "currentStep"].%X11 )
      Coil( "DB_Outputs".activeMask[11] )
   END_RUNG
   RUNG wire#powerrail
      Contact( "DB_Outputs".maskSequence[0, "currentStep"].%X12 )
      Coil( "DB_Outputs".activeMask[12] )
   END_RUNG
   RUNG wire#powerrail
      Contact( "DB_Outputs".maskSequence[0, "currentStep"].%X13 )
      Coil( "DB_Outputs".activeMask[13] )
   END_RUNG
   RUNG wire#powerrail
      Contact( "DB_Outputs".maskSequence[0, "currentStep"].%X14 )
      Coil( "DB_Outputs".activeMask[14] )
   END_RUNG
   RUNG wire#powerrail
      Contact( "DB_Outputs".maskSequence[0, "currentStep"].%X15 )
      Coil( "DB_Outputs".activeMask[15] )
   END_RUNG
   RUNG wire#powerrail
      Contact( "DB_Outputs".maskSequence[0, "currentStep"].%X16 )
      Coil( "DB_Outputs".activeMask[16] )
   END_RUNG
   RUNG wire#powerrail
      Contact( "DB_Outputs".maskSequence[0, "currentStep"].%X17 )
      Coil( "DB_Outputs".activeMask[17] )
   END_RUNG
   RUNG wire#powerrail
      Contact( "DB_Outputs".maskSequence[0, "currentStep"].%X18 )
      Coil( "DB_Outputs".activeMask[18] )
   END_RUNG
   RUNG wire#powerrail
      Contact( "DB_Outputs".maskSequence[0, "currentStep"].%X19 )
      Coil( "DB_Outputs".activeMask[19] )
   END_RUNG
   RUNG wire#powerrail
      Contact( "DB_Outputs".maskSequence[0, "currentStep"].%X20 )
      Coil( "DB_Outputs".activeMask[20] )
   END_RUNG
   RUNG wire#powerrail
      Contact( "DB_Outputs".maskSequence[0, "currentStep"].%X21 )
      Coil( "DB_Outputs".activeMask[21] )
   END_RUNG
   RUNG wire#powerrail
      Contact( "DB_Outputs".maskSequence[0, "currentStep"].%X22 )
      Coil( "DB_Outputs".activeMask[22] )
   END_RUNG
   RUNG wire#powerrail
      Contact( "DB_Outputs".maskSequence[0, "currentStep"].%X23 )
      Coil( "DB_Outputs".activeMask[23] )
   END_RUNG
   RUNG wire#powerrail
      Contact( "DB_Outputs".maskSequence[0, "currentStep"].%X24 )
      Coil( "DB_Outputs".activeMask[24] )
   END_RUNG
   RUNG wire#powerrail
      Contact( "DB_Outputs".maskSequence[0, "currentStep"].%X25 )
      Coil( "DB_Outputs".activeMask[25] )
   END_RUNG
   RUNG wire#powerrail
      Contact( "DB_Outputs".maskSequence[0, "currentStep"].%X26 )
      Coil( "DB_Outputs".activeMask[26] )
   END_RUNG
   RUNG wire#powerrail
      Contact( "DB_Outputs".maskSequence[0, "currentStep"].%X27 )
      Coil( "DB_Outputs".activeMask[27] )
   END_RUNG
   RUNG wire#powerrail
      Contact( "DB_Outputs".maskSequence[0, "currentStep"].%X28 )
      Coil( "DB_Outputs".activeMask[28] )
   END_RUNG
   RUNG wire#powerrail
      Contact( "DB_Outputs".maskSequence[0, "currentStep"].%X29 )
      Coil( "DB_Outputs".activeMask[29] )
   END_RUNG
   RUNG wire#powerrail
      Contact( "DB_Outputs".maskSequence[0, "currentStep"].%X30 )
      Coil( "DB_Outputs".activeMask[30] )
   END_RUNG
   RUNG wire#powerrail
      Contact( "DB_Outputs".maskSequence[0, "currentStep"].%X31 )
      Coil( "DB_Outputs".activeMask[31] )
   END_RUNG
   // the same network as SCL:
   "DB_Outputs".activeMask[0] := "DB_Outputs".maskSequence[0, "currentStep"].%X0;
   "DB_Outputs".activeMask[1] := "DB_Outputs".maskSequence[0, "currentStep"].%X1;
   "DB_Outputs".activeMask[2] := "DB_Outputs".maskSequence[0, "currentStep"].%X2;
   "DB_Outputs".activeMask[3] := "DB_Outputs".maskSequence[0, "currentStep"].%X3;
   "DB_Outputs".activeMask[4] := "DB_Outputs".maskSequence[0, "currentStep"].%X4;
   "DB_Outputs".activeMask[5] := "DB_Outputs".maskSequence[0, "currentStep"].%X5;
   "DB_Outputs".activeMask[6] := "DB_Outputs".maskSequence[0, "currentStep"].%X6;
   "DB_Outputs".activeMask[7] := "DB_Outputs".maskSequence[0, "currentStep"].%X7;
   "DB_Outputs".activeMask[8] := "DB_Outputs".maskSequence[0, "currentStep"].%X8;
   "DB_Outputs".activeMask[9] := "DB_Outputs".maskSequence[0, "currentStep"].%X9;
   "DB_Outputs".activeMask[10] := "DB_Outputs".maskSequence[0, "currentStep"].%X10;
   "DB_Outputs".activeMask[11] := "DB_Outputs".maskSequence[0, "currentStep"].%X11;
   "DB_Outputs".activeMask[12] := "DB_Outputs".maskSequence[0, "currentStep"].%X12;
   "DB_Outputs".activeMask[13] := "DB_Outputs".maskSequence[0, "currentStep"].%X13;
   "DB_Outputs".activeMask[14] := "DB_Outputs".maskSequence[0, "currentStep"].%X14;
   "DB_Outputs".activeMask[15] := "DB_Outputs".maskSequence[0, "currentStep"].%X15;
   "DB_Outputs".activeMask[16] := "DB_Outputs".maskSequence[0, "currentStep"].%X16;
   "DB_Outputs".activeMask[17] := "DB_Outputs".maskSequence[0, "currentStep"].%X17;
   "DB_Outputs".activeMask[18] := "DB_Outputs".maskSequence[0, "currentStep"].%X18;
   "DB_Outputs".activeMask[19] := "DB_Outputs".maskSequence[0, "currentStep"].%X19;
   "DB_Outputs".activeMask[20] := "DB_Outputs".maskSequence[0, "currentStep"].%X20;
   "DB_Outputs".activeMask[21] := "DB_Outputs".maskSequence[0, "currentStep"].%X21;
   "DB_Outputs".activeMask[22] := "DB_Outputs".maskSequence[0, "currentStep"].%X22;
   "DB_Outputs".activeMask[23] := "DB_Outputs".maskSequence[0, "currentStep"].%X23;
   "DB_Outputs".activeMask[24] := "DB_Outputs".maskSequence[0, "currentStep"].%X24;
   "DB_Outputs".activeMask[25] := "DB_Outputs".maskSequence[0, "currentStep"].%X25;
   "DB_Outputs".activeMask[26] := "DB_Outputs".maskSequence[0, "currentStep"].%X26;
   "DB_Outputs".activeMask[27] := "DB_Outputs".maskSequence[0, "currentStep"].%X27;
   "DB_Outputs".activeMask[28] := "DB_Outputs".maskSequence[0, "currentStep"].%X28;
   "DB_Outputs".activeMask[29] := "DB_Outputs".maskSequence[0, "currentStep"].%X29;
   "DB_Outputs".activeMask[30] := "DB_Outputs".maskSequence[0, "currentStep"].%X30;
   "DB_Outputs".activeMask[31] := "DB_Outputs".maskSequence[0, "currentStep"].%X31;
END_REGION
END_FUNCTION
